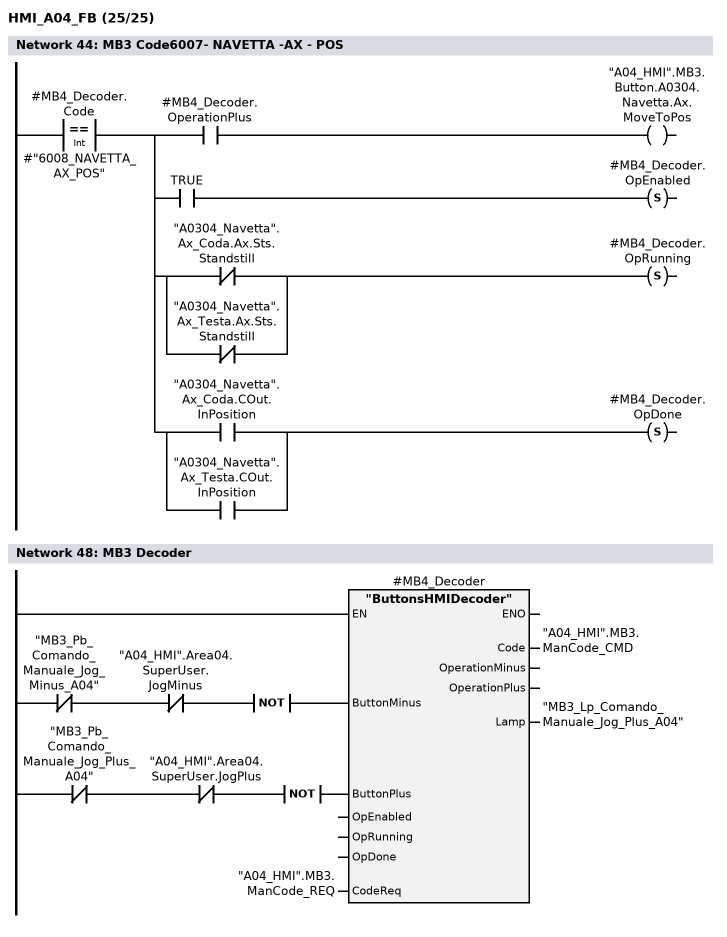
   RUNG wire#powerrail
      { S7_Templates := "SrcType := Int" } EQ_Contact(in1 := #MB4_Decoder.Code, in2 := #"6008_NAVETTA_AX_POS")
      wire#w1
      Contact( #MB4_Decoder.OperationPlus )
      Coil( "A04_HMI".MB3.Button.A0304.Navetta.Ax.MoveToPos )
   END_RUNG
   RUNG wire#w1
      Contact( TRUE )
      S_Coil( #MB4_Decoder.OpEnabled )
   END_RUNG
   RUNG wire#w1
      I_Contact( "A0304_Navetta".Ax_Coda.Ax.Sts.Standstill )
      wire#w2
      S_Coil( #MB4_Decoder.OpRunning )
   END_RUNG
   RUNG wire#w1
      I_Contact( "A0304_Navetta".Ax_Testa.Ax.Sts.Standstill )
   END_RUNG wire#w2
   RUNG wire#w1
      Contact( "A0304_Navetta".Ax_Coda.COut.InPosition )
      wire#w3
      S_Coil( #MB4_Decoder.OpDone )
   END_RUNG
   RUNG wire#w1
      Contact( "A0304_Navetta".Ax_Testa.COut.InPosition )
   END_RUNG wire#w3
   // the same network as SCL:
   #_w1 := #MB4_Decoder.Code = #"6008_NAVETTA_AX_POS";
   "A04_HMI".MB3.Button.A0304.Navetta.Ax.MoveToPos := #_w1 AND #MB4_Decoder.OperationPlus;
   IF #_w1 AND TRUE THEN #MB4_Decoder.OpEnabled := TRUE; END_IF;
   IF #_w1 AND (NOT "A0304_Navetta".Ax_Coda.Ax.Sts.Standstill OR NOT "A0304_Navetta".Ax_Testa.Ax.Sts.Standstill) THEN
       #MB4_Decoder.OpRunning := TRUE;
   END_IF;
   IF #_w1 AND ("A0304_Navetta".Ax_Coda.COut.InPosition OR "A0304_Navetta".Ax_Testa.COut.InPosition) THEN
       #MB4_Decoder.OpDone := TRUE;
   END_IF;
END_REGION

REGION Network 45: >
END_REGION

REGION Network 46: >
END_REGION

REGION Network 47: >
END_REGION

REGION Network 48: MB3 Decoder
   RUNG wire#powerrail
      #MB4_Decoder(ButtonMinus := wire#w1, ButtonPlus := wire#w2, OpEnabled :=, OpRunning :=, OpDone :=, CodeReq := "A04_HMI".MB3.ManCode_REQ, Code => "A04_HMI".MB3.ManCode_CMD, OperationMinus =>, OperationPlus =>, Lamp => "MB3_Lp_Comando_Manuale_Jog_Plus_A04")
   END_RUNG
   RUNG wire#powerrail
      I_Contact( "MB3_Pb_Comando_Manuale_Jog_Minus_A04" )
      I_Contact( "A04_HMI".Area04.SuperUser.JogMinus )
      Not()
   END_RUNG wire#w1
   RUNG wire#powerrail
      I_Contact( "MB3_Pb_Comando_Manuale_Jog_Plus_A04" )
      I_Contact( "A04_HMI".Area04.SuperUser.JogPlus )
      Not()
   END_RUNG wire#w2
   // the same network as SCL:
   #MB4_Decoder(ButtonMinus := NOT (NOT "MB3_Pb_Comando_Manuale_Jog_Minus_A04" AND NOT "A04_HMI".Area04.SuperUser.JogMinus),   // "ButtonsHMIDecoder"
                ButtonPlus := NOT (NOT "MB3_Pb_Comando_Manuale_Jog_Plus_A04" AND NOT "A04_HMI".Area04.SuperUser.JogPlus),
                CodeReq := "A04_HMI".MB3.ManCode_REQ,
                Code => "A04_HMI".MB3.ManCode_CMD,
                Lamp => "MB3_Lp_Comando_Manuale_Jog_Plus_A04");
END_REGION
END_FUNCTION_BLOCK
